FUNCTION_BLOCK newProductsOrder (* JADE WORKER *)
  (* Standard: 61499-1 *)
  (* Version 1.0, 2014-04-22, Ahmed, Fraunhofer IGD *)
  (* Compiler header: package fb.rt; *)
  (* Compiler Java Sun JDK 1.5.0 *)
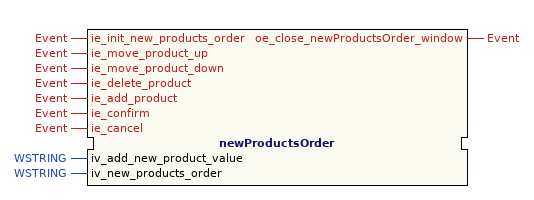
  EVENT_INPUT
    ie_init_new_products_order;
    ie_move_product_up;
    ie_move_product_down;
    ie_delete_product;
    ie_add_product;
    ie_confirm;
    ie_cancel;
  END_EVENT
  EVENT_OUTPUT
    oe_close_newProductsOrder_window;
  END_EVENT
  VAR_INPUT
    iv_add_new_product_value : WSTRING;
    iv_new_products_order : WSTRING;
  END_VAR
END_FUNCTION_BLOCK
